// TIA Portal project "ISA_P2" (V16)

(* hardware
DEVICE "PC-System_1"  SIMATIC PC station
   slot 0: "Estación PC SIMATIC"  Rail  SIMATIC PC-Station  V1.0
      slot 125: "Stationmanager"  Station_Manager  V6.0.4
   slot 1: "HMI_RT_1"  WinCC RT Advanced  6AV2 104-0xxxx-xxxx  16.0.0.0
      slot 33792: "Interfaz del equipo"  Host interface
   slot 2: "IE general_1"  IE General  IE_CP  V8.2.0
DEVICE "S7-1200 station_1"  S7-1200 Station
   slot 0: "Rack_0"  S7-1200 Rack  Rack  V1.0
   slot 1: "PLC_1"  CPU 1215C DC/DC/DC  6ES7 215-1AG40-0XB0  V4.4
*)

// ===== PLC "PLC_1"  CPU 1215C DC/DC/DC =====

VAR_GLOBAL   // PLC tag table "Tabla de variables estándar"
   "AI0" AT %IW64 : Int;
   "AQ0" AT %QW64 : Int;
   "Q0.0" AT %Q0.0 : Bool;
   "Q0.1" AT %Q0.1 : Bool;
END_VAR

DATA_BLOCK "Variables"   // DB1
{ S7_Optimized_Access := 'TRUE' }
VERSION : 0.1
   VAR
      Temp_norm : Real;   // Valor normalizado de IW64
      Temperatura : Real;   // Valor escalado de temperatura
      Potenciómetro : Int;   // Valor del potenciómetro en SCADA
      Pot_norm : Real;   // Valor normalizado del potenciómetro
   END_VAR
BEGIN
END_DATA_BLOCK

ORGANIZATION_BLOCK "Main"   // OB1, LAD, ProgramCycle
TITLE = "Main Program Sweep (Cycle)"
{ S7_Optimized_Access := 'TRUE' }
VERSION : 0.1
   VAR_INPUT
      Initial_Call : Bool;   // Initial call of this OB
      Remanence : Bool;   // =True, if remanent data are available
   END_VAR
BEGIN

REGION Network 1: Escalado Entrada IW64
   // Escalar el termómetro para que de una señal de 0 a 50ºC
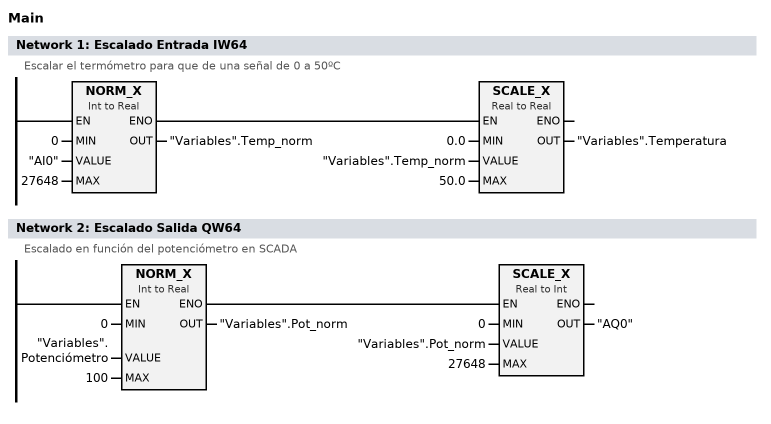
   RUNG wire#powerrail
      { S7_Templates := "[SrcType := Int, DestType := Real]" } Normalize(min := 0, value := "AI0", max := 27648, out => "Variables".Temp_norm)
      { S7_Templates := "[SrcType := Real, DestType := Real]" } Scale(min := 0.0, value := "Variables".Temp_norm, max := 50.0, out => "Variables".Temperatura)
   END_RUNG
   // the same network as SCL:
   "Variables".Temp_norm := NORM_X(MIN := 0, VALUE := "AI0", MAX := 27648);
   "Variables".Temperatura := SCALE_X(MIN := 0.0, VALUE := "Variables".Temp_norm, MAX := 50.0);
END_REGION

REGION Network 2: Escalado Salida QW64
   // Escalado en función del potenciómetro en SCADA
   RUNG wire#powerrail
      { S7_Templates := "[SrcType := Int, DestType := Real]" } Normalize(min := 0, value := "Variables".Potenciómetro, max := 100, out => "Variables".Pot_norm)
      { S7_Templates := "[SrcType := Real, DestType := Int]" } Scale(min := 0, value := "Variables".Pot_norm, max := 27648, out => "AQ0")
   END_RUNG
   // the same network as SCL:
   "Variables".Pot_norm := NORM_X(MIN := 0, VALUE := "Variables".Potenciómetro, MAX := 100);
   "AQ0" := SCALE_X(MIN := 0, VALUE := "Variables".Pot_norm, MAX := 27648);
END_REGION
END_ORGANIZATION_BLOCK

ORGANIZATION_BLOCK "Tratamiento posterior"   // OB123, LAD, ProgramCycle
TITLE = "Main Program Sweep (Cycle)"
{ S7_Optimized_Access := 'TRUE' }
VERSION : 0.1
   VAR_INPUT
      Initial_Call : Bool;   // Initial call of this OB
      Remanence : Bool;   // =True, if remanent data are available
   END_VAR
BEGIN

REGION Network 1: Salida Q0.0
   // Activar cuando la temperatura suba de 40,5ºC y desactivarla cuando baje de 35ºC
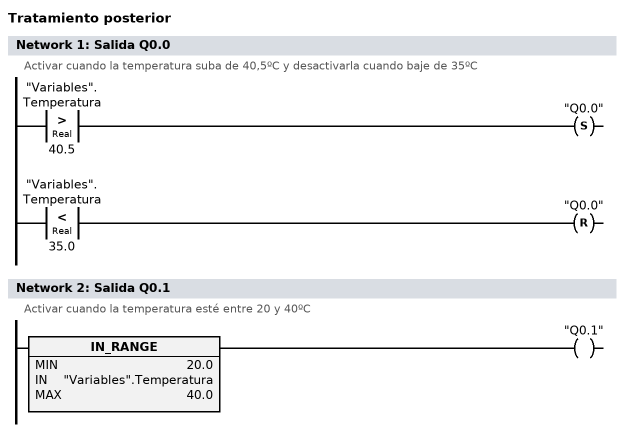
   RUNG wire#powerrail
      { S7_Templates := "SrcType := Real" } GT_Contact(in1 := "Variables".Temperatura, in2 := 40.5)
      S_Coil( "Q0.0" )
   END_RUNG
   RUNG wire#powerrail
      { S7_Templates := "SrcType := Real" } LT_Contact(in1 := "Variables".Temperatura, in2 := 35.0)
      R_Coil( "Q0.0" )
   END_RUNG
   // the same network as SCL:
   IF "Variables".Temperatura > 40.5 THEN "Q0.0" := TRUE; END_IF;
   IF "Variables".Temperatura < 35.0 THEN "Q0.0" := FALSE; END_IF;
END_REGION

REGION Network 2: Salida Q0.1
   // Activar cuando la temperatura esté entre 20 y 40ºC
   RUNG wire#powerrail
      { S7_Templates := "SrcType := Real" } InRange(min := 20.0, in := "Variables".Temperatura, max := 40.0)
      Coil( "Q0.1" )
   END_RUNG
   // the same network as SCL:
   "Q0.1" := (20.0 <= "Variables".Temperatura) AND ("Variables".Temperatura <= 40.0);
END_REGION
END_ORGANIZATION_BLOCK

(* ===== HMI "HMI_RT_1" =====
connection "HMI_Conexión_1": ETHERNET, S7_1200_OMS

HMI tags "Tabla de variables estándar"
   "Variables_Temperatura" : Real = PLC Variables.Temperatura, 1 s
   "Variables_Potenciómetro" : Int = PLC Variables.Potenciómetro, 1 s

screen "Imagen_1" 800x600
   IOField "Campo ES_1" at 213,113 size 62x32; FormatPattern 99.9
      ProcessValue <- "Variables_Temperatura"
   TextField "Campo de texto_1" at 124,117 size 63x22; Text 'Tº (ºC):'
   Slider "Deslizador_1" at 507,82 size 80x230; Caption 'SIMATIC'
      ProcessValue <- "Variables_Potenciómetro"
*)